TYPE Track_Segment :			// all values formatted from Track_Segment_Raw
STRUCT
	iID : INT;					// track number
	rStart : REAL;				// local start of barcode
	rEnd : REAL;				// local end of barcode
	rAbsoluteStart : REAL;		// x_position
	rAbsoluteEnd : REAL;		// x_position + length
END_STRUCT
END_TYPE

(* stored: Version 1.1.0.1
   DUT Track_Segment: Id {0d8d06af-89ea-472f-bd49-85dc9ba4a40c} *)
